LIN {X 0,Y 90.479,Z 349.119,A -85,B 0,C 180,E1 -30592.051,E2 -30592.051} C_VEL
LIN {X 0,Y 99.07,Z 339.253,A -85,B 0,C 180,E1 -30593.303,E2 -30593.303} C_VEL
LIN {X 0,Y 106.82,Z 328.134,A -85,B 0,C 180,E1 -30594.348,E2 -30594.348} C_VEL
LIN {X 0,Y 112.874,Z 317.228,A -85,B 0,C 180,E1 -30595.03,E2 -30595.03} C_VEL
LIN {X 0,Y 117.95,Z 305.457,A -85,B 0,C 180,E1 -30595.631,E2 -30595.631} C_VEL
LIN {X 0,Y 120.879,Z 296.506,A -85,B 0,C 180,E1 -30596.097,E2 -30596.097} C_VEL
LIN {X 0,Y 121.085,Z 295.11,A -85,B 0,C 180,E1 -30600,E2 -30600} C_VEL
LIN {X 0,Y 120.982,Z 296.479,A -85,B 0,C 180,E1 -30603.444,E2 -30603.444} C_VEL
LIN {X 0,Y 116.631,Z 309.235,A -85,B 0,C 180,E1 -30603.837,E2 -30603.837} C_VEL
LIN {X 0,Y 110.998,Z 321.287,A -85,B 0,C 180,E1 -30604.248,E2 -30604.248} C_VEL
LIN {X 0,Y 104.045,Z 332.826,A -85,B 0,C 180,E1 -30604.899,E2 -30604.899} C_VEL
LIN {X 0,Y 96.237,Z 343.222,A -85,B 0,C 180,E1 -30605.716,E2 -30605.716} C_VEL
LIN {X 0,Y 88.454,Z 351.723,A -85,B 0,C 180,E1 -30606.688,E2 -30606.688} C_VEL
LIN {X 0,Y 78.146,Z 360.944,A -85,B 0,C 180,E1 -30608.385,E2 -30608.385} C_VEL
LIN {X 0,Y 67.955,Z 368.37,A -85,B 0,C 180,E1 -30610.72,E2 -30610.72} C_VEL
LIN {X 0,Y 56.786,Z 374.958,A -85,B 0,C 180,E1 -30614.331,E2 -30614.331} C_VEL
LIN {X 0,Y 48.157,Z 379.063,A -85,B 0,C 180,E1 -30618.438,E2 -30618.438} C_VEL
LIN {X 0,Y 38.79,Z 382.675,A -85,B 0,C 180,E1 -30625.042,E2 -30625.042} C_VEL
LIN {X 0,Y 32.93,Z 384.537,A -85,B 0,C 180,E1 -30631.373,E2 -30631.373} C_VEL
LIN {X 0,Y 23.47,Z 386.954,A -85,B 0,C 180,E1 -30653.198,E2 -30653.198} C_VEL
LIN {X 0,Y 20.737,Z 387.577,A -85,B 0,C 180,E1 -30670.179,E2 -30670.179} C_VEL
LIN {X 0,Y 20.034,Z 387.8,A -85,B 0,C 180,E1 -30689.989,E2 -30689.989} C_VEL
LIN {X 0,Y 20.742,Z 387.556,A -85,B 0,C 180,E1 -30709.794,E2 -30709.794} C_VEL
LIN {X 0,Y 23.476,Z 386.92,A -85,B 0,C 180,E1 -30726.768,E2 -30726.768} C_VEL
LIN {X 0,Y 32.923,Z 384.466,A -85,B 0,C 180,E1 -30748.62,E2 -30748.62} C_VEL
LIN {X 0,Y 41.842,Z 381.497,A -85,B 0,C 180,E1 -30757.473,E2 -30757.473} C_VEL
LIN {X 0,Y 51.378,Z 377.49,A -85,B 0,C 180,E1 -30763.224,E2 -30763.224} C_VEL
LIN {X 0,Y 62.914,Z 371.333,A -85,B 0,C 180,E1 -30767.789,E2 -30767.789} C_VEL
LIN {X 0,Y 73.024,Z 364.623,A -85,B 0,C 180,E1 -30770.545,E2 -30770.545} C_VEL
LIN {X 0,Y 83.286,Z 356.314,A -85,B 0,C 180,E1 -30772.501,E2 -30772.501} C_VEL
LIN {X 0,Y 91.901,Z 347.788,A -85,B 0,C 180,E1 -30773.774,E2 -30773.774} C_VEL
LIN {X 0,Y 100.558,Z 337.263,A -85,B 0,C 180,E1 -30774.799,E2 -30774.799} C_VEL
LIN {X 0,Y 107.511,Z 326.85,A -85,B 0,C 180,E1 -30775.449,E2 -30775.449} C_VEL
LIN {X 0,Y 113.637,Z 315.345,A -85,B 0,C 180,E1 -30775.958,E2 -30775.958} C_VEL
LIN {X 0,Y 118.458,Z 303.414,A -85,B 0,C 180,E1 -30776.339,E2 -30776.339} C_VEL
LIN {X 0,Y 120.699,Z 296.235,A -85,B 0,C 180,E1 -30776.587,E2 -30776.587} C_VEL
LIN {X 0,Y 120.822,Z 294.795,A -85,B 0,C 180,E1 -30780,E2 -30780} C_VEL
LIN {X 0,Y 120.598,Z 296.295,A -85,B 0,C 180,E1 -30784.056,E2 -30784.056} C_VEL
LIN {X 0,Y 116.337,Z 308.748,A -85,B 0,C 180,E1 -30784.607,E2 -30784.607} C_VEL
LIN {X 0,Y 111.148,Z 320,A -85,B 0,C 180,E1 -30785.227,E2 -30785.227} C_VEL
LIN {X 0,Y 104.24,Z 331.597,A -85,B 0,C 180,E1 -30786.057,E2 -30786.057} C_VEL
LIN {X 0,Y 96.489,Z 342.019,A -85,B 0,C 180,E1 -30787.091,E2 -30787.091} C_VEL
LIN {X 0,Y 88.78,Z 350.531,A -85,B 0,C 180,E1 -30788.324,E2 -30788.324} C_VEL
LIN {X 0,Y 79.95,Z 358.659,A -85,B 0,C 180,E1 -30790.126,E2 -30790.126} C_VEL
LIN {X 0,Y 70.189,Z 366.02,A -85,B 0,C 180,E1 -30792.526,E2 -30792.526} C_VEL
LIN {X 0,Y 61.861,Z 371.252,A -85,B 0,C 180,E1 -30795.071,E2 -30795.071} C_VEL
LIN {X 0,Y 52.034,Z 376.324,A -85,B 0,C 180,E1 -30799.024,E2 -30799.024} C_VEL
LIN {X 0,Y 45.598,Z 379.084,A -85,B 0,C 180,E1 -30802.835,E2 -30802.835} C_VEL
LIN {X 0,Y 40.414,Z 380.964,A -85,B 0,C 180,E1 -30805.719,E2 -30805.719} C_VEL
LIN {X 0,Y 31.149,Z 383.5,A -85,B 0,C 180,E1 -30809.691,E2 -30809.691} C_VEL
LIN {X 0,Y 23.717,Z 385.003,A -85,B 0,C 180,E1 -30814.81,E2 -30814.81} C_VEL
LIN {X 0,Y 18.738,Z 385.809,A -85,B 0,C 180,E1 -30823.296,E2 -30823.296} C_VEL
LIN {X 0,Y 17.376,Z 385.968,A -85,B 0,C 180,E1 -30827.801,E2 -30827.801} C_VEL
LIN {X 0,Y 13.306,Z 386.582,A -85,B 0,C 180,E1 -30870.016,E2 -30870.016} C_VEL
LIN {X 0,Y 14.877,Z 386.387,A -85,B 0,C 180,E1 -30898.207,E2 -30898.207} C_VEL
LIN {X 0,Y 24.415,Z 384.839,A -85,B 0,C 180,E1 -30929.736,E2 -30929.736} C_VEL
LIN {X 0,Y 30.468,Z 383.485,A -85,B 0,C 180,E1 -30937.334,E2 -30937.334} C_VEL
LIN {X 0,Y 40.155,Z 380.618,A -85,B 0,C 180,E1 -30944.303,E2 -30944.303} C_VEL
LIN {X 0,Y 50.164,Z 376.73,A -85,B 0,C 180,E1 -30948.741,E2 -30948.741} C_VEL
LIN {X 0,Y 60.401,Z 371.702,A -85,B 0,C 180,E1 -30951.521,E2 -30951.521} C_VEL
LIN {X 0,Y 70.714,Z 365.369,A -85,B 0,C 180,E1 -30953.671,E2 -30953.671} C_VEL
LIN {X 0,Y 81.089,Z 357.45,A -85,B 0,C 180,E1 -30955.368,E2 -30955.368} C_VEL
LIN {X 0,Y 91.516,Z 347.597,A -85,B 0,C 180,E1 -30956.727,E2 -30956.727} C_VEL
LIN {X 0,Y 100.241,Z 337.23,A -85,B 0,C 180,E1 -30957.573,E2 -30957.573} C_VEL
LIN {X 0,Y 107.231,Z 326.966,A -85,B 0,C 180,E1 -30958.212,E2 -30958.212} C_VEL
LIN {X 0,Y 113.835,Z 314.74,A -85,B 0,C 180,E1 -30958.751,E2 -30958.751} C_VEL
LIN {X 0,Y 118.643,Z 302.891,A -85,B 0,C 180,E1 -30959.147,E2 -30959.147} C_VEL
LIN {X 0,Y 118.938,Z 302.018,A -85,B 0,C 180,E1 -30959.548,E2 -30959.548} C_VEL
LIN {X 0,Y 118.929,Z 302.069,A -85,B 0,C 180,E1 -30960,E2 -30960} C_VEL
LIN {X 0,Y 118.661,Z 302.882,A -85,B 0,C 180,E1 -30960.233,E2 -30960.233} C_VEL
LIN {X 0,Y 113.853,Z 314.777,A -85,B 0,C 180,E1 -30960.491,E2 -30960.491} C_VEL
LIN {X 0,Y 108.066,Z 325.709,A -85,B 0,C 180,E1 -30960.722,E2 -30960.722} C_VEL
LIN {X 0,Y 100.172,Z 337.458,A -85,B 0,C 180,E1 -30961.181,E2 -30961.181} C_VEL
LIN {X 0,Y 91.411,Z 347.889,A -85,B 0,C 180,E1 -30961.8,E2 -30961.8} C_VEL
LIN {X 0,Y 82.666,Z 356.337,A -85,B 0,C 180,E1 -30962.592,E2 -30962.592} C_VEL
LIN {X 0,Y 72.203,Z 364.597,A -85,B 0,C 180,E1 -30963.861,E2 -30963.861} C_VEL
LIN {X 0,Y 61.805,Z 371.263,A -85,B 0,C 180,E1 -30965.715,E2 -30965.715} C_VEL
LIN {X 0,Y 49.792,Z 377.365,A -85,B 0,C 180,E1 -30968.856,E2 -30968.856} C_VEL
LIN {X 0,Y 39.666,Z 381.337,A -85,B 0,C 180,E1 -30972.952,E2 -30972.952} C_VEL
LIN {X 0,Y 29.847,Z 384.278,A -85,B 0,C 180,E1 -30979.614,E2 -30979.614} C_VEL
LIN {X 0,Y 18.274,Z 386.695,A -85,B 0,C 180,E1 -30999.701,E2 -30999.701} C_VEL
LIN {X 0,Y 14.24,Z 387.317,A -85,B 0,C 180,E1 -31020.411,E2 -31020.411} C_VEL
LIN {X 0,Y 12.936,Z 387.54,A -85,B 0,C 180,E1 -31049.984,E2 -31049.984} C_VEL
LIN {X 0,Y 14.244,Z 387.295,A -85,B 0,C 180,E1 -31079.548,E2 -31079.548} C_VEL
LIN {X 0,Y 18.275,Z 386.659,A -85,B 0,C 180,E1 -31100.257,E2 -31100.257} C_VEL
LIN {X 0,Y 29.84,Z 384.205,A -85,B 0,C 180,E1 -31120.381,E2 -31120.381} C_VEL
LIN {X 0,Y 39.659,Z 381.236,A -85,B 0,C 180,E1 -31127.046,E2 -31127.046} C_VEL
LIN {X 0,Y 49.788,Z 377.228,A -85,B 0,C 180,E1 -31131.122,E2 -31131.122} C_VEL
LIN {X 0,Y 61.798,Z 371.07,A -85,B 0,C 180,E1 -31134.284,E2 -31134.284} C_VEL
LIN {X 0,Y 72.196,Z 364.36,A -85,B 0,C 180,E1 -31136.141,E2 -31136.141} C_VEL
LIN {X 0,Y 82.658,Z 356.051,A -85,B 0,C 180,E1 -31137.414,E2 -31137.414} C_VEL
LIN {X 0,Y 91.404,Z 347.526,A -85,B 0,C 180,E1 -31138.206,E2 -31138.206} C_VEL
LIN {X 0,Y 100.164,Z 337,A -85,B 0,C 180,E1 -31138.842,E2 -31138.842} C_VEL
LIN {X 0,Y 107.181,Z 326.586,A -85,B 0,C 180,E1 -31139.236,E2 -31139.236} C_VEL
LIN {X 0,Y 113.488,Z 314.803,A -85,B 0,C 180,E1 -31139.546,E2 -31139.546} C_VEL
LIN {X 0,Y 118.372,Z 302.686,A -85,B 0,C 180,E1 -31139.788,E2 -31139.788} C_VEL
LIN {X 0,Y 118.686,Z 301.739,A -85,B 0,C 180,E1 -31140,E2 -31140} C_VEL
LIN {X 0,Y 118.677,Z 301.738,A -85,B 0,C 180,E1 -31140.525,E2 -31140.525} C_VEL
LIN {X 0,Y 118.014,Z 303.704,A -85,B 0,C 180,E1 -31140.949,E2 -31140.949} C_VEL
LIN {X 0,Y 113.081,Z 315.568,A -85,B 0,C 180,E1 -31141.334,E2 -31141.334} C_VEL
LIN {X 0,Y 106.353,Z 327.825,A -85,B 0,C 180,E1 -31141.923,E2 -31141.923} C_VEL
LIN {X 0,Y 98.493,Z 339.081,A -85,B 0,C 180,E1 -31142.655,E2 -31142.655} C_VEL
LIN {X 0,Y 89.774,Z 349.019,A -85,B 0,C 180,E1 -31143.544,E2 -31143.544} C_VEL
LIN {X 0,Y 81.087,Z 357.156,A -85,B 0,C 180,E1 -31144.707,E2 -31144.707} C_VEL
LIN {X 0,Y 70.719,Z 365.122,A -85,B 0,C 180,E1 -31146.42,E2 -31146.42} C_VEL
LIN {X 0,Y 60.406,Z 371.513,A -85,B 0,C 180,E1 -31148.56,E2 -31148.56} C_VEL
LIN {X 0,Y 50.17,Z 376.584,A -85,B 0,C 180,E1 -31151.336,E2 -31151.336} C_VEL
LIN {X 0,Y 40.161,Z 380.51,A -85,B 0,C 180,E1 -31155.768,E2 -31155.768} C_VEL
LIN {X 0,Y 30.484,Z 383.407,A -85,B 0,C 180,E1 -31162.774,E2 -31162.774} C_VEL
LIN {X 0,Y 24.416,Z 384.786,A -85,B 0,C 180,E1 -31170.304,E2 -31170.304} C_VEL
LIN {X 0,Y 17.376,Z 385.968,A -85,B 0,C 180,E1 -31187.801,E2 -31187.801} C_VEL
LIN {X 0,Y 14.894,Z 386.328,A -85,B 0,C 180,E1 -31198.65,E2 -31198.65} C_VEL
LIN {X 0,Y 11.64,Z 386.625,A -85,B 0,C 180,E1 -31220.321,E2 -31220.321} C_VEL
LIN {X 0,Y 13.191,Z 386.324,A -85,B 0,C 180,E1 -31288.545,E2 -31288.545} C_VEL
LIN {X 0,Y 18.826,Z 385.58,A -85,B 0,C 180,E1 -31303.248,E2 -31303.248} C_VEL
LIN {X 0,Y 19.749,Z 385.383,A -85,B 0,C 180,E1 -31304.299,E2 -31304.299} C_VEL
LIN {X 0,Y 28.496,Z 383.744,A -85,B 0,C 180,E1 -31310.619,E2 -31310.619} C_VEL
LIN {X 0,Y 38.84,Z 380.877,A -85,B 0,C 180,E1 -31314.431,E2 -31314.431} C_VEL
LIN {X 0,Y 49.273,Z 376.988,A -85,B 0,C 180,E1 -31316.855,E2 -31316.855} C_VEL
LIN {X 0,Y 61.52,Z 370.98,A -85,B 0,C 180,E1 -31318.454,E2 -31318.454} C_VEL
LIN {X 0,Y 63.272,Z 369.978,A -85,B 0,C 180,E1 -31318.648,E2 -31318.648} C_VEL
LIN {X 0,Y 63.266,Z 369.989,A -85,B 0,C 180,E1 -31318.901,E2 -31318.901} C_VEL
LIN {X 0,Y 53.161,Z 375.306,A -85,B 0,C 180,E1 -31320,E2 -31320} C_VEL
LIN {X 0,Y 42.192,Z 379.853,A -85,B 0,C 180,E1 -31321.817,E2 -31321.817} C_VEL
LIN {X 0,Y 35.211,Z 382.157,A -85,B 0,C 180,E1 -31323.547,E2 -31323.547} C_VEL
LIN {X 0,Y 28.265,Z 384.019,A -85,B 0,C 180,E1 -31325.891,E2 -31325.891} C_VEL
LIN {X 0,Y 14.769,Z 386.434,A -85,B 0,C 180,E1 -31337.837,E2 -31337.837} C_VEL
LIN {X 0,Y 8.788,Z 387.058,A -85,B 0,C 180,E1 -31356.856,E2 -31356.856} C_VEL
LIN {X 0,Y 5.826,Z 387.281,A -85,B 0,C 180,E1 -31409.964,E2 -31409.964} C_VEL
LIN {X 0,Y 8.786,Z 387.035,A -85,B 0,C 180,E1 -31463.078,E2 -31463.078} C_VEL
LIN {X 0,Y 21.4,Z 385.371,A -85,B 0,C 180,E1 -31490.077,E2 -31490.077} C_VEL
LIN {X 0,Y 28.257,Z 383.945,A -85,B 0,C 180,E1 -31494.107,E2 -31494.107} C_VEL
LIN {X 0,Y 38.689,Z 380.974,A -85,B 0,C 180,E1 -31497.425,E2 -31497.425} C_VEL
LIN {X 0,Y 49.194,Z 376.965,A -85,B 0,C 180,E1 -31499.398,E2 -31499.398} C_VEL
LIN {X 0,Y 61.498,Z 370.808,A -85,B 0,C 180,E1 -31500.914,E2 -31500.914} C_VEL
LIN {X 0,Y 63.259,Z 369.793,A -85,B 0,C 180,E1 -31501.096,E2 -31501.096} C_VEL
LIN {X 0,Y 63.268,Z 369.778,A -85,B 0,C 180,E1 -31501.457,E2 -31501.457} C_VEL
LIN {X 0,Y 52.65,Z 375.315,A -85,B 0,C 180,E1 -31502.726,E2 -31502.726} C_VEL
LIN {X 0,Y 42.305,Z 379.558,A -85,B 0,C 180,E1 -31504.679,E2 -31504.679} C_VEL
LIN {X 0,Y 35.375,Z 381.826,A -85,B 0,C 180,E1 -31506.67,E2 -31506.67} C_VEL
LIN {X 0,Y 28.498,Z 383.667,A -85,B 0,C 180,E1 -31509.488,E2 -31509.488} C_VEL
LIN {X 0,Y 21.719,Z 385.045,A -85,B 0,C 180,E1 -31513.936,E2 -31513.936} C_VEL
LIN {X 0,Y 9.243,Z 386.623,A -85,B 0,C 180,E1 -31540.541,E2 -31540.541} C_VEL
LIN {X 0,Y 6.211,Z 386.841,A -85,B 0,C 180,E1 -31590.034,E2 -31590.034} C_VEL
LIN {X 0,Y 9.248,Z 386.646,A -85,B 0,C 180,E1 -31639.491,E2 -31639.491} C_VEL
LIN {X 0,Y 19.749,Z 385.383,A -85,B 0,C 180,E1 -31664.299,E2 -31664.299} C_VEL
LIN {X 0,Y 21.906,Z 387.364,A -85,B 0,C 180,E1 -31666.262,E2 -31666.262} C_VEL
LIN {X 0,Y 21.906,Z 600,A -85,B 0,C 180,E1 -31666.262,E2 -31666.262} C_VEL
LIN {X 0,Y 21.906,Z 600,A -85,B 0,C 180,E1 -31666.262,E2 -31666.262}

QRS_NEXT_CUT()

QRS_NEXT()
QRS_HOME()

END
